FUNCTION SendErrorMessage : BOOL
VAR_INPUT
	message : REFERENCE TO FB_TcMessage;
	position : STRING;
	POUNAME : STRING;
END_VAR
VAR
	_tmpStr : STRING;
END_VAR

message.ipArguments.AddString(__POUNAME());
_tmpStr := formatPosition(__POSITION());
message.ipArguments.AddString(_tmpStr);
message.Send(0);

SendErrorMessage := TRUE;
RETURN;

END_FUNCTION

(* stored: Version 1.1.0.1
   POU SendErrorMessage: Id {350d1a04-5c84-4457-af14-48add8ed2a1f}, SpecialFunc None *)
